PROGRAM PRG_GameSession
VAR
    T_Ronde : TON;
END_VAR

IF (Biertjes >= 3) AND NOT SpelGestart THEN
    SpelGestart := TRUE;
END_IF

IF SpelGestart AND (Ronde < 10) THEN
    T_Ronde(IN := TRUE, PT := T#4S);

    IF T_Ronde.Q THEN
        Ronde := Ronde + 1;
        T_Ronde(IN := FALSE);
    END_IF
END_IF

IF Ronde >= 10 THEN
    AvondKlaar := TRUE;
END_IF

END_PROGRAM

(* stored: Version 1.1.0.1, ProductVersion 3.1.4024.15
   POU PRG_GameSession: Id {84fb9743-b88f-4f77-87db-d0a8d16619d2}, SpecialFunc None *)
